// SIMATIC S7-200 SMART project (STEP 7-Micro/WIN SMART), CPU ST40

SYMBOL_TABLE 表格 1
Marker           VD2000   // 标志位
END_SYMBOL_TABLE

SYMBOL_TABLE 系统符号
Always_On        SM0.0    // 始终接通
END_SYMBOL_TABLE

ORGANIZATION_BLOCK MAIN:OB1
TITLE=程序注释
VAR
NUB:INT;	// LW0 
END_VAR
BEGIN
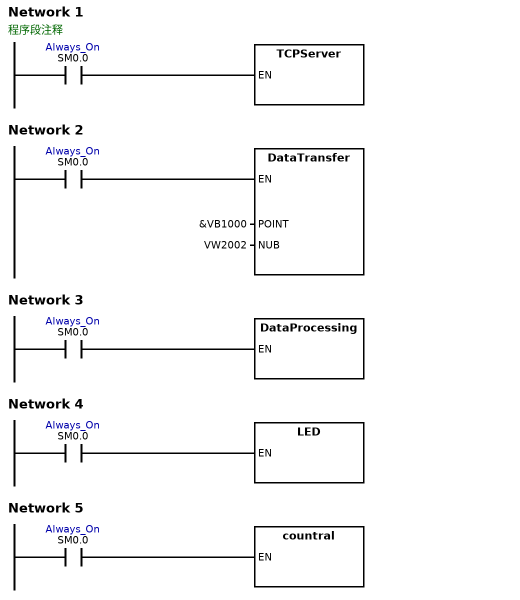
Network 1
// 程序段注释
LD     Always_On:SM0.0
CALL   TCPServer:SBR50
Network 2
LD     Always_On:SM0.0
CALL   DataTransfer:SBR53, &VB1000, VW2002
Network 3
LD     Always_On:SM0.0
CALL   DataProcessing:SBR54
Network 4
LD     Always_On:SM0.0
CALL   LED:SBR11
Network 5
LD     Always_On:SM0.0
CALL   countral:SBR0
END_ORGANIZATION_BLOCK

SUBROUTINE_BLOCK countral:SBR0
TITLE=子程序注释
BEGIN
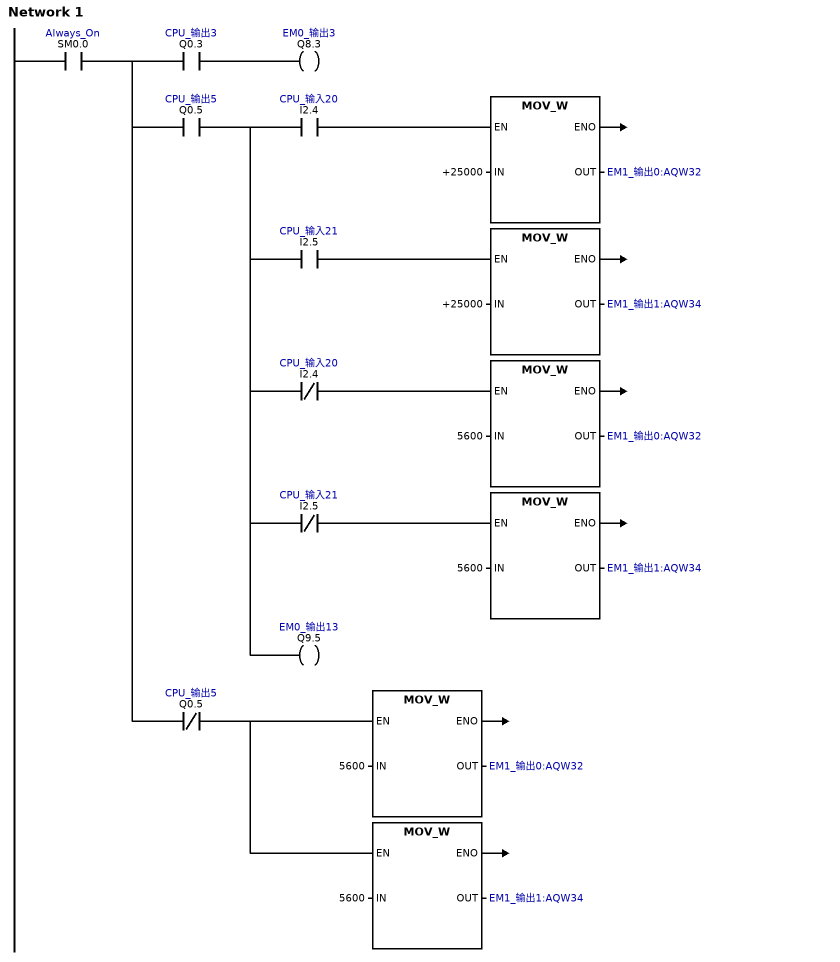
Network 1
LD     Always_On:SM0.0
LPS
A      CPU_输出3:Q0.3
=      EM0_输出3:Q8.3
LRD
A      CPU_输出5:Q0.5
LPS
A      CPU_输入20:I2.4
MOVW   +25000, EM1_输出0:AQW32
LRD
A      CPU_输入21:I2.5
MOVW   +25000, EM1_输出1:AQW34
LRD
AN     CPU_输入20:I2.4
MOVW   5600, EM1_输出0:AQW32
LRD
AN     CPU_输入21:I2.5
MOVW   5600, EM1_输出1:AQW34
LPP
=      EM0_输出13:Q9.5
LPP
AN     CPU_输出5:Q0.5
MOVW   5600, EM1_输出0:AQW32
MOVW   5600, EM1_输出1:AQW34
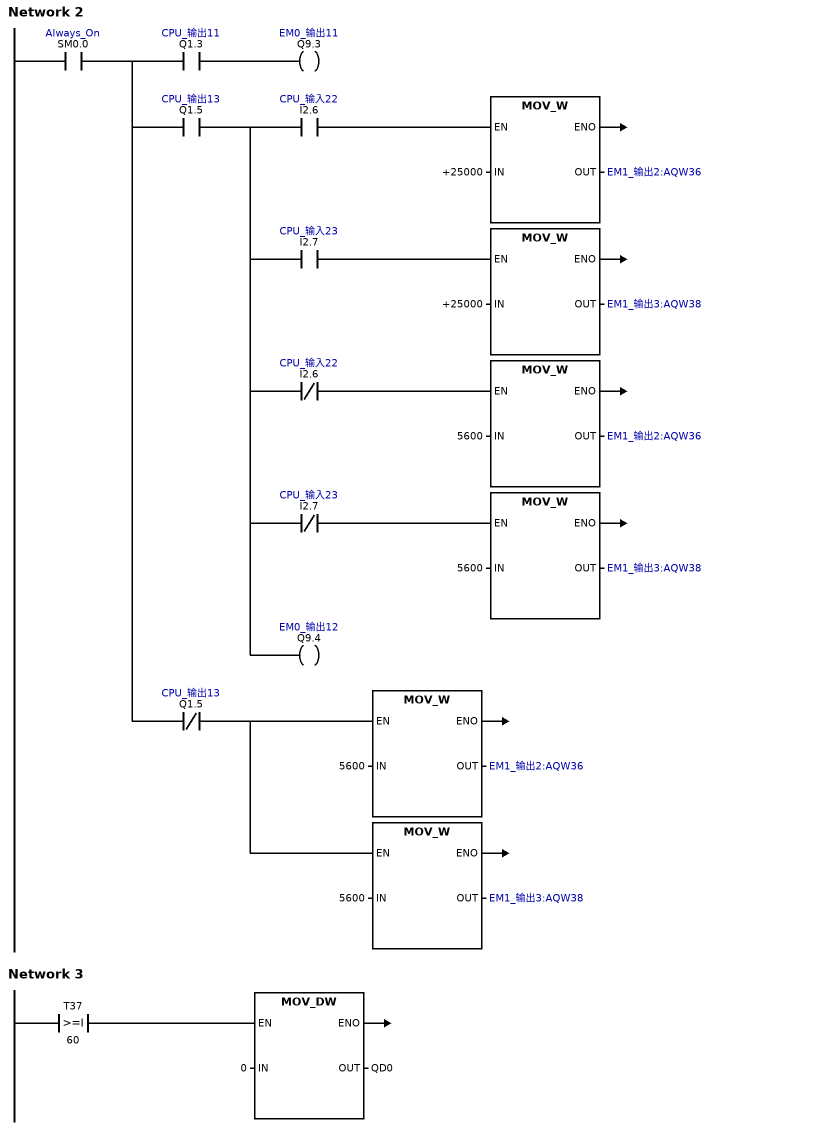
Network 2
LD     Always_On:SM0.0
LPS
A      CPU_输出11:Q1.3
=      EM0_输出11:Q9.3
LRD
A      CPU_输出13:Q1.5
LPS
A      CPU_输入22:I2.6
MOVW   +25000, EM1_输出2:AQW36
LRD
A      CPU_输入23:I2.7
MOVW   +25000, EM1_输出3:AQW38
LRD
AN     CPU_输入22:I2.6
MOVW   5600, EM1_输出2:AQW36
LRD
AN     CPU_输入23:I2.7
MOVW   5600, EM1_输出3:AQW38
LPP
=      EM0_输出12:Q9.4
LPP
AN     CPU_输出13:Q1.5
MOVW   5600, EM1_输出2:AQW36
MOVW   5600, EM1_输出3:AQW38
Network 3
LDW>=  T37, 60
MOVD   0, QD0
END_SUBROUTINE_BLOCK

// SBR3: protected block, not included

// SBR4: protected block, not included

// SBR5: protected block, not included

// SBR6: protected block, not included

SUBROUTINE_BLOCK output:SBR10
TITLE=子程序注释
BEGIN
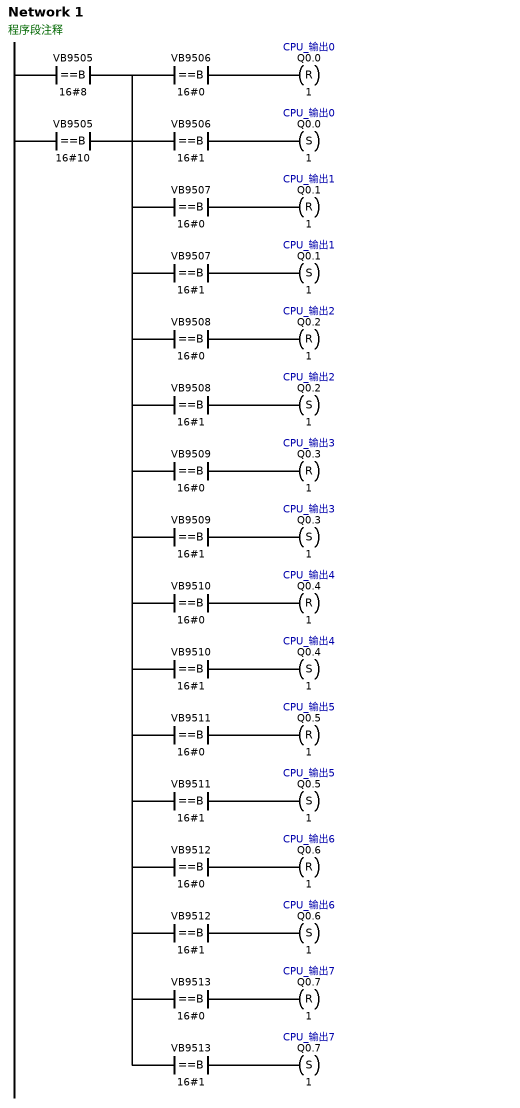
Network 1
// 程序段注释
LDB=   VB9505, 16#8
OB=    VB9505, 16#10
LPS
AB=    VB9506, 16#0
R      CPU_输出0:Q0.0, 1
LRD
AB=    VB9506, 16#1
S      CPU_输出0:Q0.0, 1
LRD
AB=    VB9507, 16#0
R      CPU_输出1:Q0.1, 1
LRD
AB=    VB9507, 16#1
S      CPU_输出1:Q0.1, 1
LRD
AB=    VB9508, 16#0
R      CPU_输出2:Q0.2, 1
LRD
AB=    VB9508, 16#1
S      CPU_输出2:Q0.2, 1
LRD
AB=    VB9509, 16#0
R      CPU_输出3:Q0.3, 1
LRD
AB=    VB9509, 16#1
S      CPU_输出3:Q0.3, 1
LRD
AB=    VB9510, 16#0
R      CPU_输出4:Q0.4, 1
LRD
AB=    VB9510, 16#1
S      CPU_输出4:Q0.4, 1
LRD
AB=    VB9511, 16#0
R      CPU_输出5:Q0.5, 1
LRD
AB=    VB9511, 16#1
S      CPU_输出5:Q0.5, 1
LRD
AB=    VB9512, 16#0
R      CPU_输出6:Q0.6, 1
LRD
AB=    VB9512, 16#1
S      CPU_输出6:Q0.6, 1
LRD
AB=    VB9513, 16#0
R      CPU_输出7:Q0.7, 1
LPP
AB=    VB9513, 16#1
S      CPU_输出7:Q0.7, 1
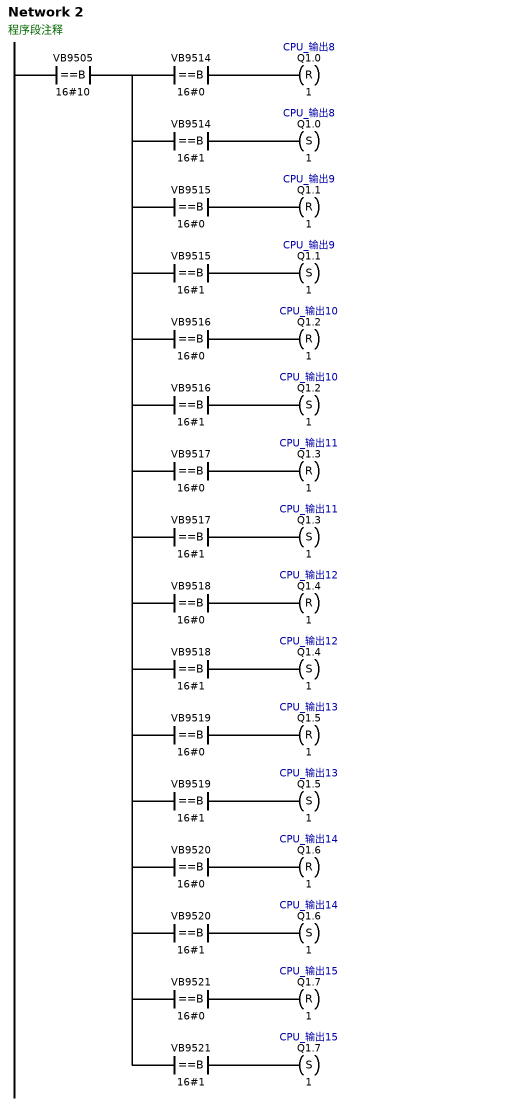
Network 2
// 程序段注释
LDB=   VB9505, 16#10
LPS
AB=    VB9514, 16#0
R      CPU_输出8:Q1.0, 1
LRD
AB=    VB9514, 16#1
S      CPU_输出8:Q1.0, 1
LRD
AB=    VB9515, 16#0
R      CPU_输出9:Q1.1, 1
LRD
AB=    VB9515, 16#1
S      CPU_输出9:Q1.1, 1
LRD
AB=    VB9516, 16#0
R      CPU_输出10:Q1.2, 1
LRD
AB=    VB9516, 16#1
S      CPU_输出10:Q1.2, 1
LRD
AB=    VB9517, 16#0
R      CPU_输出11:Q1.3, 1
LRD
AB=    VB9517, 16#1
S      CPU_输出11:Q1.3, 1
LRD
AB=    VB9518, 16#0
R      CPU_输出12:Q1.4, 1
LRD
AB=    VB9518, 16#1
S      CPU_输出12:Q1.4, 1
LRD
AB=    VB9519, 16#0
R      CPU_输出13:Q1.5, 1
LRD
AB=    VB9519, 16#1
S      CPU_输出13:Q1.5, 1
LRD
AB=    VB9520, 16#0
R      CPU_输出14:Q1.6, 1
LRD
AB=    VB9520, 16#1
S      CPU_输出14:Q1.6, 1
LRD
AB=    VB9521, 16#0
R      CPU_输出15:Q1.7, 1
LPP
AB=    VB9521, 16#1
S      CPU_输出15:Q1.7, 1
END_SUBROUTINE_BLOCK

SUBROUTINE_BLOCK LED:SBR11
TITLE=
BEGIN
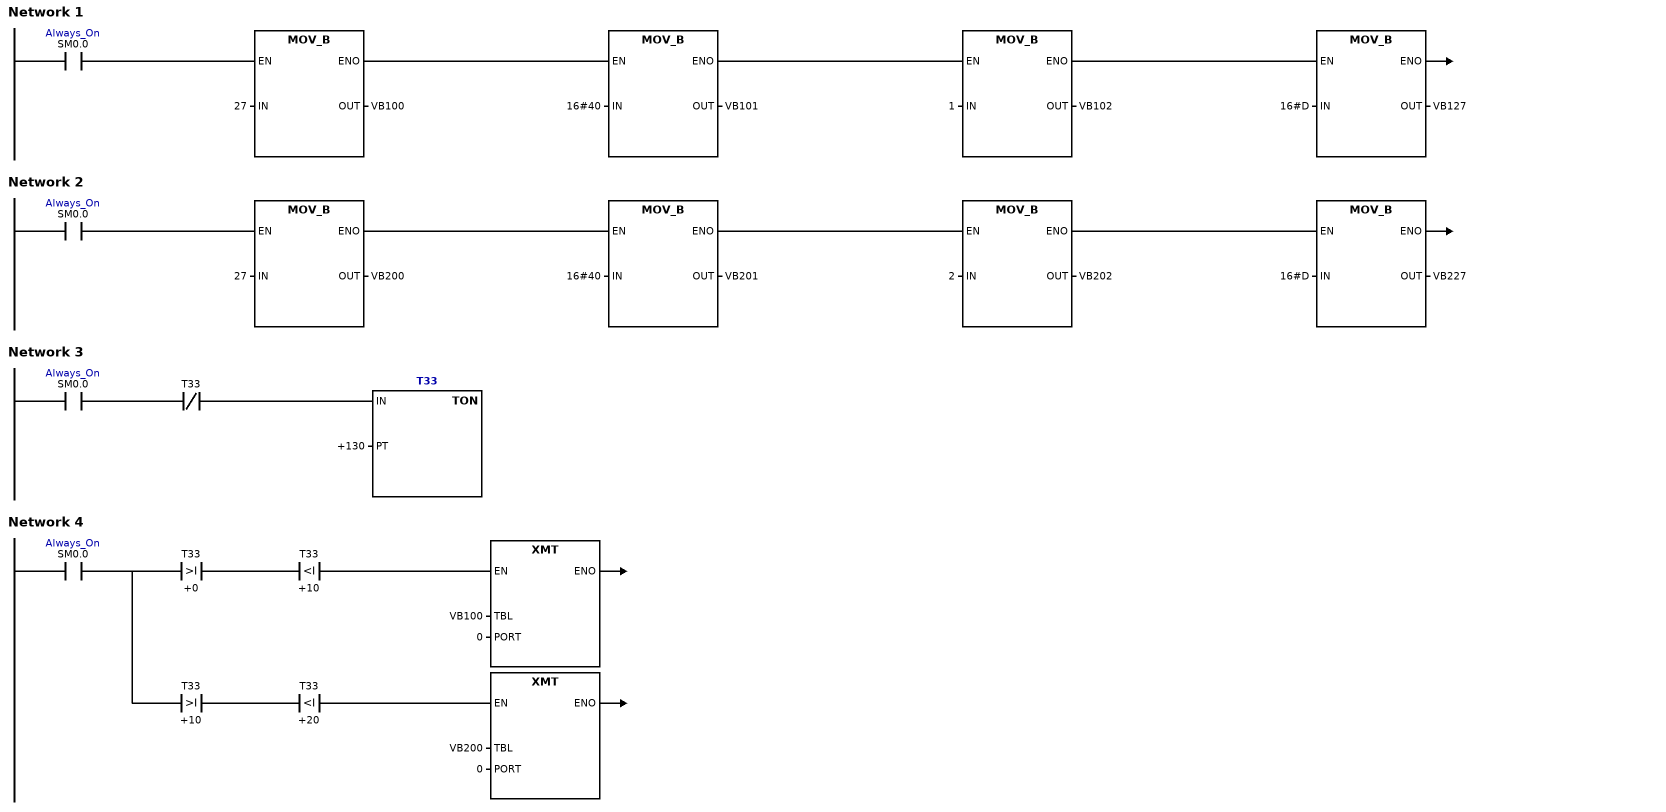
Network 1
LD     Always_On:SM0.0
MOVB   27, VB100
AENO
MOVB   16#40, VB101
AENO
MOVB   1, VB102
AENO
MOVB   16#D, VB127
Network 2
LD     Always_On:SM0.0
MOVB   27, VB200
AENO
MOVB   16#40, VB201
AENO
MOVB   2, VB202
AENO
MOVB   16#D, VB227
Network 3
LD     Always_On:SM0.0
AN     T33
TON    T33, +130
Network 4
LD     Always_On:SM0.0
LPS
AW>    T33, +0
AW<    T33, +10
XMT    VB100, 0
LPP
AW>    T33, +10
AW<    T33, +20
XMT    VB200, 0
END_SUBROUTINE_BLOCK

SUBROUTINE_BLOCK XORCheck:SBR12
TITLE=子程序注释
VAR_INPUT
NO1:DWORD;	// LD0 
NO2:DWORD;	// LD4 
NUB:WORD;	// LW8 
END_VAR
VAR_OUTPUT
RESULT:BYTE;	// LB10 
END_VAR
VAR
COUNT:WORD;	// LW11 
TEMP:BYTE;	// LB13 
END_VAR
BEGIN
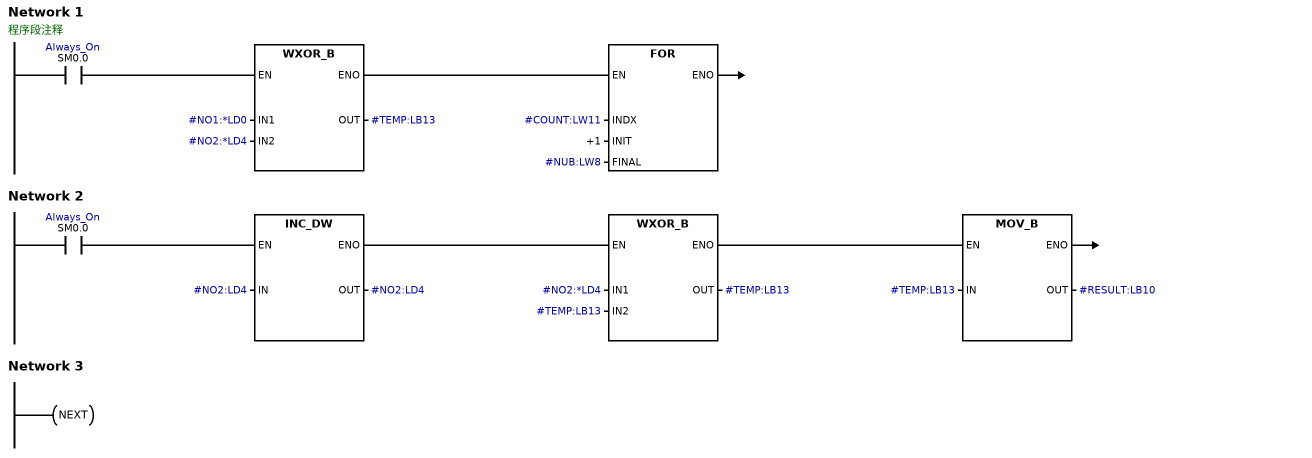
Network 1
// 程序段注释
LD     Always_On:SM0.0
MOVB   *#NO1:LD0, #TEMP:LB13
AENO
XORB   *#NO2:LD4, #TEMP:LB13
AENO
FOR    #COUNT:LW11, +1, #NUB:LW8
Network 2
LD     Always_On:SM0.0
INCD   #NO2:LD4
AENO
XORB   *#NO2:LD4, #TEMP:LB13
AENO
MOVB   #TEMP:LB13, #RESULT:LB10
Network 3
NEXT
END_SUBROUTINE_BLOCK

// SBR50: protected block, not included

// SBR51: protected block, not included

// SBR52: protected block, not included

// SBR53: protected block, not included

// SBR54: protected block, not included
